{attribute 'qualified_only'}
{attribute 'strict'}
{attribute 'to_string'}
TYPE EnvironmentErrorEnum :
(
no_error	:=	0	,//	No error detected
not_connected	:=	1	,//	A command was requested prior to opening the driver
invalid_state	:=	2	,//	An invalid command was requested
io_error	:=	3	,//	IO error HW board
unknown_error	:=	4	,//	Unknown / Network error
emergency_error	:=	666	//	




	
);
END_TYPE

(* stored: Version 1.1.0.1, ProductVersion 3.1.4024.11
   DUT EnvironmentErrorEnum: Id {a8bfc5ec-49ca-443a-8160-daf57725c2cb} *)
